% RSLogix 500 project DIGITAL_TANK_PUMP_CONTROL.RSS, saved by version 8.30.00.16 %
PROJECT "UNTITLED"    % processor: Bul.1763 MicroLogix 1100 Series B %

PROGRAM FILES
  LAD 2 "MAIN"  4 rungs
  LAD 3 "ALARM"  7 rungs
  LAD 4 "IO"  9 rungs  % IO %
  LAD 5 "CONTROL"  6 rungs

DATA FILES
  O0 OUTPUT  4 elements
  I1 INPUT  6 elements
  S2 STATUS  66 elements
  B3 BINARY  1 elements
  T4 TIMER  5 elements
  C5 COUNTER  1 elements
  R6 CONTROL  1 elements
  N7 INTEGER  1 elements
  F8 FLOAT  1 elements

LADDER 2 "MAIN"
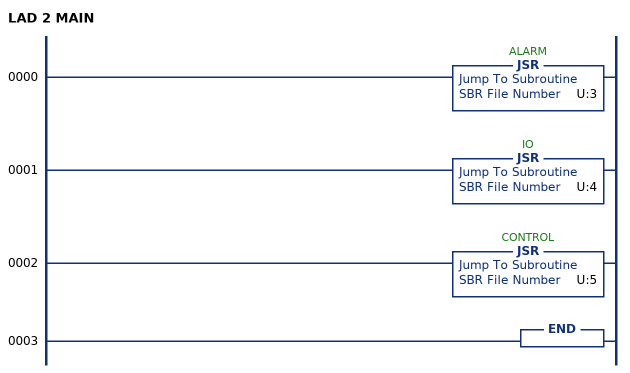
% Rung: 0 %
SOR JSR U:3 EOR
%   U:3  "ALARM" %
% Rung: 1 %
SOR JSR U:4 EOR
%   U:4  "IO" %
% Rung: 2 %
SOR JSR U:5 EOR
%   U:5  "CONTROL" %
% Rung: 3 %
SOR END EOR

LADDER 3 "ALARM"
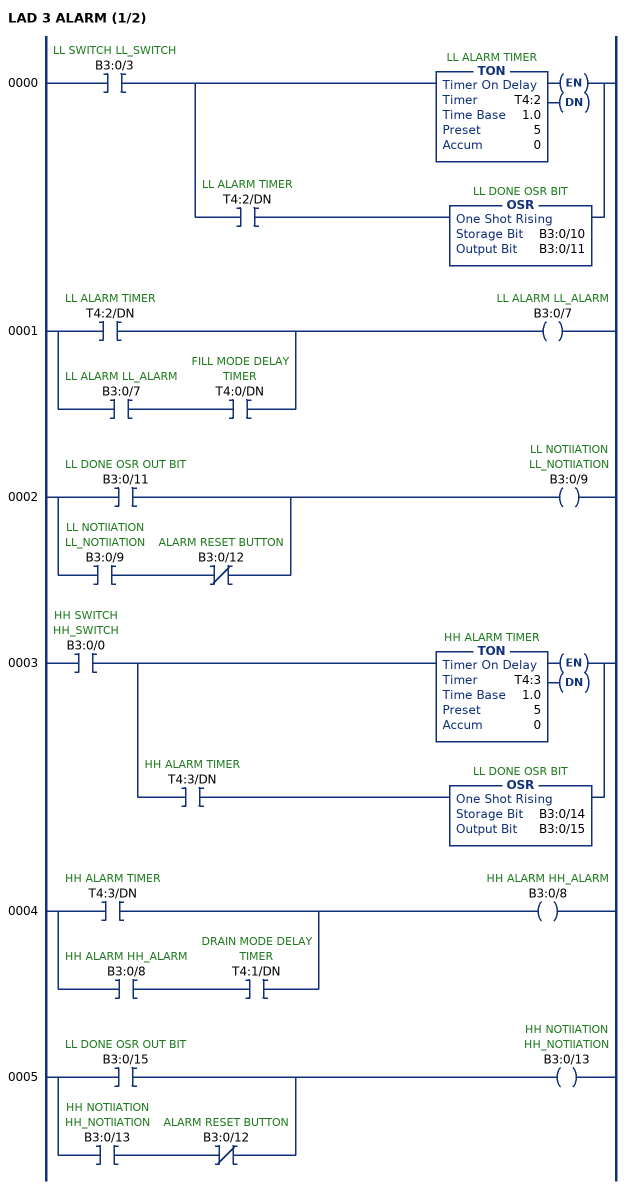
% Rung: 0 %
SOR XIC B3:0/3 BST TON T4:2 1.0 5 0 NXB XIC T4:2/DN OSR B3:0/10 B3:0/11 BND EOR
%   B3:0/3  LL_SWITCH  "LL SWITCH" %
%   T4:2  "LL ALARM TIMER" %
%   B3:0/10  "LL DONE OSR BIT" %
%   B3:0/11  "LL DONE OSR OUT BIT" %
% Rung: 1 %
SOR BST XIC T4:2/DN NXB XIC B3:0/7 XIC T4:0/DN BND OTE B3:0/7 EOR
%   T4:2  "LL ALARM TIMER" %
%   B3:0/7  LL_ALARM  "LL ALARM" %
%   T4:0  "FILL MODE DELAY TIMER" %
% Rung: 2 %
SOR BST XIC B3:0/11 NXB XIC B3:0/9 XIO B3:0/12 BND OTE B3:0/9 EOR
%   B3:0/11  "LL DONE OSR OUT BIT" %
%   B3:0/9  LL_NOTIIATION  "LL NOTIIATION" %
%   B3:0/12  "ALARM RESET BUTTON" %
% Rung: 3 %
SOR XIC B3:0/0 BST TON T4:3 1.0 5 0 NXB XIC T4:3/DN OSR B3:0/14 B3:0/15 BND EOR
%   B3:0/0  HH_SWITCH  "HH SWITCH" %
%   T4:3  "HH ALARM TIMER" %
%   B3:0/14  "LL DONE OSR BIT" %
%   B3:0/15  "LL DONE OSR OUT BIT" %
% Rung: 4 %
SOR BST XIC T4:3/DN NXB XIC B3:0/8 XIC T4:1/DN BND OTE B3:0/8 EOR
%   T4:3  "HH ALARM TIMER" %
%   B3:0/8  HH_ALARM  "HH ALARM" %
%   T4:1  "DRAIN MODE DELAY TIMER" %
% Rung: 5 %
SOR BST XIC B3:0/15 NXB XIC B3:0/13 XIO B3:0/12 BND OTE B3:0/13 EOR
%   B3:0/15  "LL DONE OSR OUT BIT" %
%   B3:0/13  HH_NOTIIATION  "HH NOTIIATION" %
%   B3:0/12  "ALARM RESET BUTTON" %

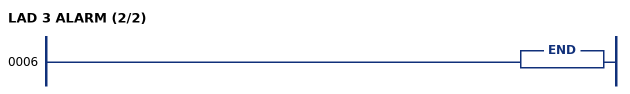
% Rung: 6 %
SOR END EOR

LADDER 4 "IO"    % IO %
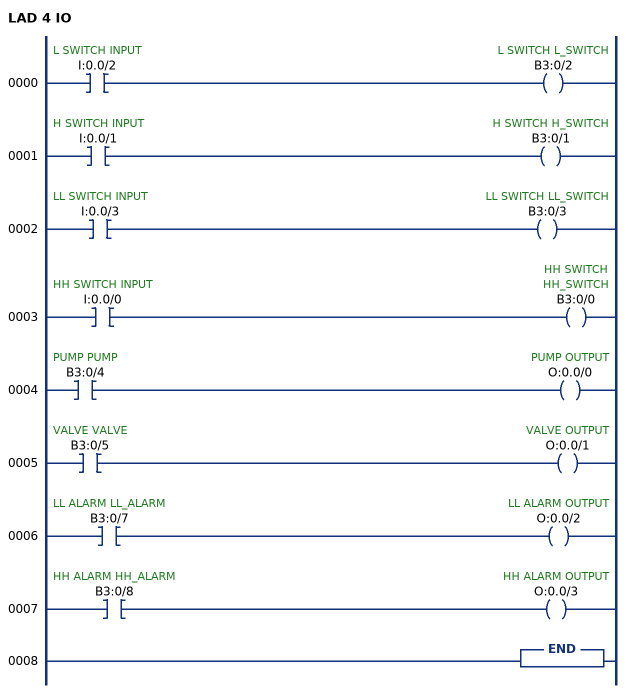
% Rung: 0 %
SOR XIC I:0.0/2 OTE B3:0/2 EOR
%   I:0.0/2  "L SWITCH INPUT" %
%   B3:0/2  L_SWITCH  "L SWITCH" %
% Rung: 1 %
SOR XIC I:0.0/1 OTE B3:0/1 EOR
%   I:0.0/1  "H SWITCH INPUT" %
%   B3:0/1  H_SWITCH  "H SWITCH" %
% Rung: 2 %
SOR XIC I:0.0/3 OTE B3:0/3 EOR
%   I:0.0/3  "LL SWITCH INPUT" %
%   B3:0/3  LL_SWITCH  "LL SWITCH" %
% Rung: 3 %
SOR XIC I:0.0/0 OTE B3:0/0 EOR
%   I:0.0/0  "HH SWITCH INPUT" %
%   B3:0/0  HH_SWITCH  "HH SWITCH" %
% Rung: 4 %
SOR XIC B3:0/4 OTE O:0.0/0 EOR
%   B3:0/4  PUMP  "PUMP" %
%   O:0.0/0  "PUMP OUTPUT" %
% Rung: 5 %
SOR XIC B3:0/5 OTE O:0.0/1 EOR
%   B3:0/5  VALVE  "VALVE" %
%   O:0.0/1  "VALVE OUTPUT" %
% Rung: 6 %
SOR XIC B3:0/7 OTE O:0.0/2 EOR
%   B3:0/7  LL_ALARM  "LL ALARM" %
%   O:0.0/2  "LL ALARM OUTPUT" %
% Rung: 7 %
SOR XIC B3:0/8 OTE O:0.0/3 EOR
%   B3:0/8  HH_ALARM  "HH ALARM" %
%   O:0.0/3  "HH ALARM OUTPUT" %
% Rung: 8 %
SOR END EOR

LADDER 5 "CONTROL"
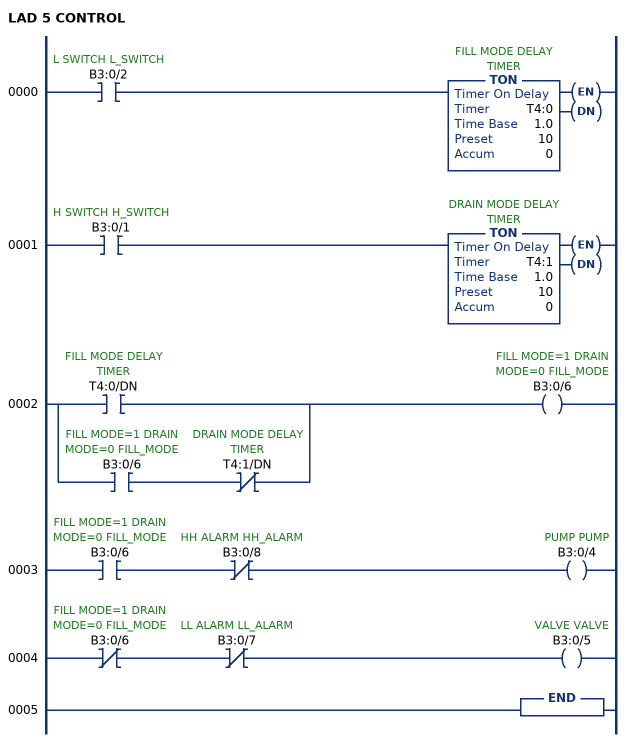
% Rung: 0 %
SOR XIC B3:0/2 TON T4:0 1.0 10 0 EOR
%   B3:0/2  L_SWITCH  "L SWITCH" %
%   T4:0  "FILL MODE DELAY TIMER" %
% Rung: 1 %
SOR XIC B3:0/1 TON T4:1 1.0 10 0 EOR
%   B3:0/1  H_SWITCH  "H SWITCH" %
%   T4:1  "DRAIN MODE DELAY TIMER" %
% Rung: 2 %
SOR BST XIC T4:0/DN NXB XIC B3:0/6 XIO T4:1/DN BND OTE B3:0/6 EOR
%   T4:0  "FILL MODE DELAY TIMER" %
%   B3:0/6  FILL_MODE  "FILL MODE=1 DRAIN MODE=0" %
%   T4:1  "DRAIN MODE DELAY TIMER" %
% Rung: 3 %
SOR XIC B3:0/6 XIO B3:0/8 OTE B3:0/4 EOR
%   B3:0/6  FILL_MODE  "FILL MODE=1 DRAIN MODE=0" %
%   B3:0/8  HH_ALARM  "HH ALARM" %
%   B3:0/4  PUMP  "PUMP" %
% Rung: 4 %
SOR XIO B3:0/6 XIO B3:0/7 OTE B3:0/5 EOR
%   B3:0/6  FILL_MODE  "FILL MODE=1 DRAIN MODE=0" %
%   B3:0/7  LL_ALARM  "LL ALARM" %
%   B3:0/5  VALVE  "VALVE" %
% Rung: 5 %
SOR END EOR

DATA TABLE (non-zero values as saved)
DATA T4
% .PRE .ACC %
% T4:0 % 10 0
% T4:1 % 10 0
% T4:2 % 5 0
% T4:3 % 5 0
